// TIA Portal V20 export
DATA_BLOCK "QDAS_WritePLCData"   // DB10001
{ S7_Optimized_Access := 'FALSE' }
// stored: AutoNumber false, InstanceOfName typeWritePLCData, InstanceOfType UDT
"typeWritePLCData"
   // VAR
   //    processData : Bool;
   //    spareOut_1 : Bool;
   //    spareOut_2 : Bool;
   //    spareOut_3 : Bool;
   //    spareOut_4 : Bool;
   //    spareOut_5 : Bool;
   //    spareOut_6 : Bool;
   //    spareOut_7 : Bool;
   //    "type" : Int;
   //    module : Int;
   //    machine : DInt;
   //    fixture : Int;
   //    pun : Array[0..31] of Char;
   //    unWinderInfeed : "typeStationDataUnwidnerInfeed";
   //    reelCutInspection : "typeStationDataReelCutInspection";
   // END_VAR
BEGIN
END_DATA_BLOCK
